FUNCTION_BLOCK Heater_control
VAR_INPUT
	terminalResistance: INT;
	desiredTemp: LREAL;
	calibrationValues: ARRAY [1..6] OF LREAL;
	maxTemp: LREAL;
END_VAR
VAR_OUTPUT
	PWM_out: BOOL;
	temperatureSensor: LREAL;
	TooHot: BOOL;
END_VAR
VAR
	fbGetTemperature: FB_GetTemperature;
	
	realTemp: LREAL;
	temperature :LREAL;
	error: LREAL; // E(k)
	previousError: LREAL; // E(k-1)
	integral: LREAL;
	derivative: LREAL;
	cycleTime: LREAL;
	controlSignal: LREAL;
	PWM: FB_PWM;
	FB_GETCURTASKINDEX:GETCURTASKINDEX;
	PID : FB_CTRL_PID;
	
	PID_params : ST_CTRL_PID_PARAMS := ( tCtrlCycleTime := T#1MS,  tTaskCycleTime:= T#1MS,fKp := 40, tTn := T#1MS ,tTv := T#1MS,  tTd := T#1M );
	
	Kp : LREAL := 120;
	Ki : LREAL := 1.5;
	Kd : LREAL := 45;
	
END_VAR

IF fbGetTemperature.temperatureSensor < maxTemp THEN
	fbGetTemperature(terminalResistance:= (10*INT_TO_REAL(terminalResistance)), calibrationValues:= calibrationValues, temperatureSensor=> temperatureSensor);// weerstand naar temperatuur conversie
	
	error := desiredTemp - temperatureSensor;
	FB_GETCURTASKINDEX();
	cycleTime := (UDINT_TO_LREAL(_TaskInfo[FB_GETCURTASKINDEX.index].CycleTime)/ 10_000_000);
	//integral := integral + error * cycleTime;
	derivative := (error - previousError) / cycleTime;
	controlSignal := (Kp * error  + Kd * derivative); //+ Ki * integral
	
	
	IF (controlSignal > 0 ) THEN
		PWM( dutyCycle := controlSignal);	
	ELSE 
		PWM(dutyCycle := 0);
	END_IF
	
	PWM_out := PWM.state; 
	previousError := error;
ELSE 
	PWM_out := FALSE;
END_IF

IF fbGetTemperature.temperatureSensor > 40 THEN
	TooHot:= TRUE;
ELSE
	TooHot:= FALSE;
END_IF

END_FUNCTION_BLOCK

(* stored: Version 1.1.0.1, ProductVersion 3.1.4024.9
   POU Heater_control: Id {dd38d42a-bd3b-456e-a2fc-9f69da39d4fa}, SpecialFunc None *)
